// SIMATIC S7-200 project (STEP 7-Micro/WIN), CPU 221 REL 01.10

SYMBOL_TABLE USER1
start            I0.0
stopp            I0.1
END_SYMBOL_TABLE

ORGANIZATION_BLOCK MAIN:OB1
TITLE=PROGRAM COMMENTS
BEGIN
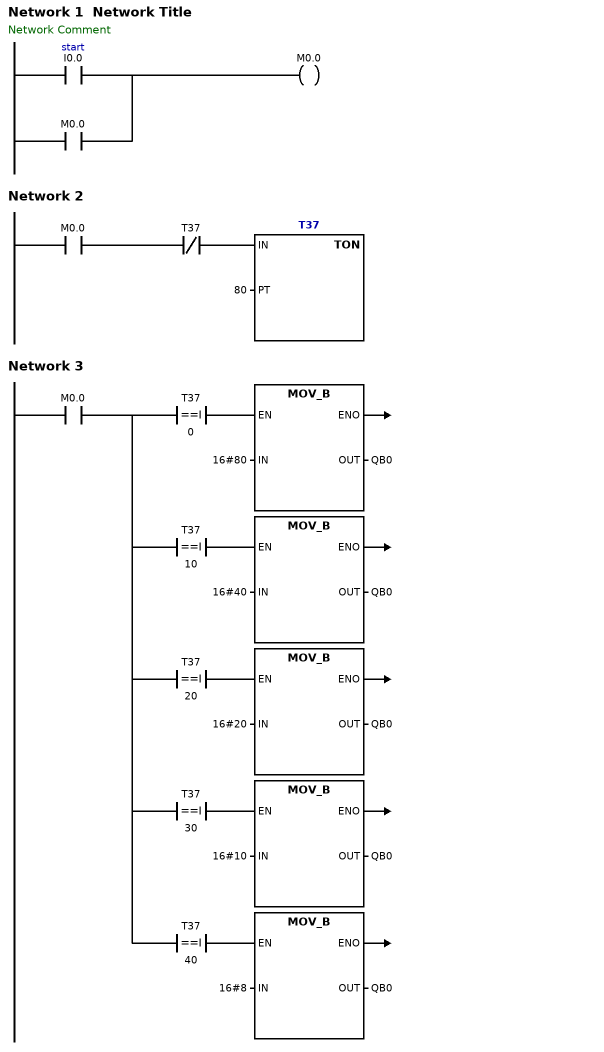
Network 1 // Network Title
// Network Comment
// (network saved uncompiled; LAD cells follow)
// row 0: c0 -| |- start:I0.0 v  c1 --  c2 -( ) M0.0
// row 1: c0 -| |- M0.0 ^
Network 2
// (network saved uncompiled; LAD cells follow)
// row 0: c0 -| |- M0.0  c1 -|/|- T37  c2 [TON T37 IN:=power@row0, PT:=80]
// row 1: c2 [box]
Network 3
// (network saved uncompiled; LAD cells follow)
// row 0: c0 -| |- M0.0 v  c1 -|==I|- T37, 0  c2 [MOV_B EN:=power@row0, IN:=16#80, ENO=>power, OUT=>QB0]  c3 ->
// row 1: c0 ^v  c2 [box]
// row 2: c0 ^v  c1 -|==I|- T37, 10  c2 [MOV_B EN:=power@row2, IN:=16#40, ENO=>power, OUT=>QB0]  c3 ->
// row 3: c0 ^v  c2 [box]
// row 4: c0 ^v  c1 -|==I|- T37, 20  c2 [MOV_B EN:=power@row4, IN:=16#20, ENO=>power, OUT=>QB0]  c3 ->
// row 5: c0 ^v  c2 [box]
// row 6: c0 ^v  c1 -|==I|- T37, 30  c2 [MOV_B EN:=power@row6, IN:=16#10, ENO=>power, OUT=>QB0]  c3 ->
// row 7: c0 ^v  c2 [box]
// row 8: c0 ^  c1 -|==I|- T37, 40  c2 [MOV_B EN:=power@row8, IN:=16#8, ENO=>power, OUT=>QB0]  c3 ->
// row 9: c2 [box]
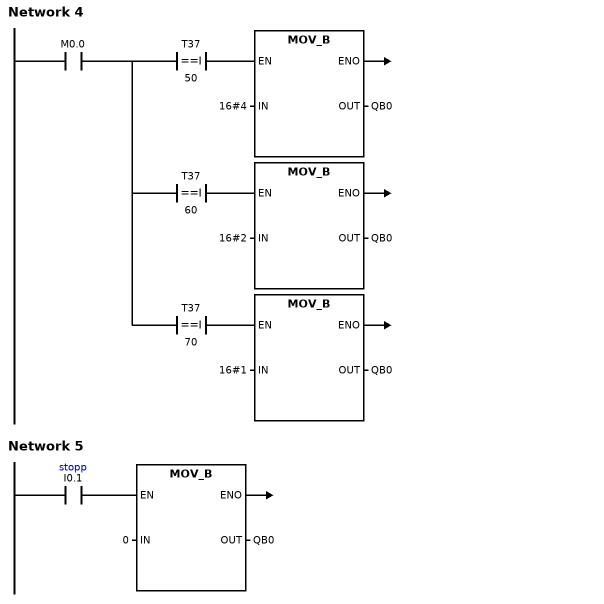
Network 4
// (network saved uncompiled; LAD cells follow)
// row 0: c0 -| |- M0.0 v  c1 -|==I|- T37, 50  c2 [MOV_B EN:=power@row0, IN:=16#4, ENO=>power, OUT=>QB0]  c3 ->
// row 1: c0 ^v  c2 [box]
// row 2: c0 ^v  c1 -|==I|- T37, 60  c2 [MOV_B EN:=power@row2, IN:=16#2, ENO=>power, OUT=>QB0]  c3 ->
// row 3: c0 ^v  c2 [box]
// row 4: c0 ^  c1 -|==I|- T37, 70  c2 [MOV_B EN:=power@row4, IN:=16#1, ENO=>power, OUT=>QB0]  c3 ->
// row 5: c2 [box]
Network 5
// (network saved uncompiled; LAD cells follow)
// row 0: c0 -| |- stopp:I0.1  c1 [MOV_B EN:=power@row0, IN:=0, ENO=>power, OUT=>QB0]  c2 ->
// row 1: c1 [box]
END_ORGANIZATION_BLOCK
